(* PLC project  *)

CONFIGURATION Empty_Module_3
END_CONFIGURATION
